Fanuc KAREL source: CNV_REAL_STR.kl

PROGRAM T
%NOLOCKGROUP
VAR
 v0 : REAL
 v1 : INTEGER
 v2 : INTEGER
 v3 : STRING[40]
BEGIN
 CNV_REAL_STR(v0, v1, v2, v3)
END T
